(* IEC 61131-3 sources: RL_MAR/experiments/comparison/autoplc/results/gpt-4o_20260511_211137/med_76, 1 file *)

(* ---- med_76_3.st ---- *)
FUNCTION_BLOCK MultimediaArtInstallationControl
    VAR_INPUT
        MotionSensor : BOOL; (* Motion detection input *)
        AudioTrack : BOOL; (* Selected audio track *)
        VisualContent : BOOL; (* Selected visual content *)
    END_VAR
    VAR_OUTPUT
        LightingControl : BOOL; (* Lighting control output *)
        AudioControl : BOOL; (* Audio playback control *)
        VisualControl : BOOL; (* Visual display control *)
    END_VAR
    VAR
        ActivationTimer : INT; (* Timer for activation duration *)
        SafetyCheckPassed : BOOL; (* Safety check status *)
    END_VAR

    // Initialization
    LightingControl := FALSE;
    AudioControl := FALSE;
    VisualControl := FALSE;
    ActivationTimer := 0;
    SafetyCheckPassed := TRUE;

    // Main Control Logic
    IF MotionSensor THEN
        // Active State Logic
        IF SafetyCheckPassed THEN
            LightingControl := TRUE;
            AudioControl := TRUE;
            VisualControl := TRUE;

            // Increment Activation Timer
            IF ActivationTimer < 300 THEN
                ActivationTimer := ActivationTimer + 1;
            END_IF
        ELSE
            // Safety Protocols Violation
            LightingControl := FALSE;
            AudioControl := FALSE;
            VisualControl := FALSE;
        END_IF
    ELSE
        // Idle State Logic
        LightingControl := FALSE;
        AudioControl := FALSE;
        VisualControl := FALSE;
        ActivationTimer := 0;
    END_IF

    // Safety Protocols
    SafetyCheckPassed := CheckSafety;

END_FUNCTION_BLOCK

FUNCTION CheckSafety : BOOL
    VAR
        PowerUsage : INT; (* Simulated power usage value *)
        SystemCheck : BOOL; (* Simulated system check status *)
    END_VAR

    // Simulate power usage and system check
    PowerUsage := 50; // Example value, should be replaced with actual measurement
    SystemCheck := TRUE; // Example value, should be replaced with actual check

    // Safety conditions
    IF (PowerUsage < 100) AND SystemCheck THEN
        CheckSafety := TRUE;
    ELSE
        CheckSafety := FALSE;
    END_IF
END_FUNCTION
